// TIA Portal V20 export
TYPE "typeSequenceControlNode_GRnR"
// stored: Namespace Unit1.Em8
   STRUCT
      jobs : "LAF_typeJobs";
      sequence : "LAF_typeSequence";
      selectJobStatus { S7_SetPoint := 'True'} : Array[0..10] of "LAF_typeJobStatus";
      "step" : "LER_typeStep";
      jobInterface : "Unit1.Em8.typeSequenceControlNodeJobInterface_GRnR";
   END_STRUCT;
   // // "step".action1[101] : Step[101] : JOB[1] Condition
   // // "step".action1[110] : Step[110] : Hipot & Thickness Z-Axis Wait Pos
   // // "step".action1[111] : Step[111] : Servo Press Reference Home Pos
   // // "step".action1[120] : Step[120] : Tab Contactor Open
   // // "step".action1[121] : Step[121] : Tab Contactor Backward
   // // "step".action1[130] : Step[130] : Stage Lift Up
   // // "step".action1[140] : Step[140] : Spare
   // // "step".action1[150] : Step[150] : Stage Lift Down
   // // "step".action1[170] : Step[170] : Spare
   // // "step".action1[190] : Step[190] : JOB[1] Step End
   // // "step".action1[201] : Step[201] : JOB[2] Condition
   // // "step".action1[210] : Step[210] : Hipot & Thickness Loading Request => Transfer PP Left
   // // "step".action1[220] : Step[220] : Spare
   // // "step".action1[230] : Step[230] : Stage Lift Up
   // // "step".action1[240] : Step[240] : Hipot & Thickness Loading Check => Transfer PP Left
   // // "step".action1[250] : Step[250] : Spare
   // // "step".action1[290] : Step[290] : JOB[2] Step End
   // // "step".action1[301] : Step[301] : JOB[3] Condition
   // // "step".action1[310] : Step[310] : Stage Lift Down
   // // "step".action1[311] : Step[311] : Stage JR Detection Check
   // // "step".action1[320] : Step[320] : Spare
   // // "step".action1[330] : Step[330] : Press Start
   // // "step".action1[331] : Step[331] : Press Result
   // // "step".action1[340] : Step[340] : Thickness Z-Axis Thickness Ready Pos, Tab Forward
   // // "step".action1[341] : Step[341] : Thickness Z-Axis Measuring Thickness Pos, Tab Contactor Close
   // // "step".action1[350] : Step[350] : Thickness Start
   // // "step".action1[351] : Step[351] : Thickness Result
   // // "step".action1[352] : Step[352] : Thickness Z-Axis Wait Pos
   // // "step".action1[360] : Step[360] : Hipot Start
   // // "step".action1[361] : Step[361] : Hipot Result
   // // "step".action1[362] : Step[362] : Tab Contactor Open
   // // "step".action1[363] : Step[363] : Tab Contactor Backward
   // // "step".action1[380] : Step[380] : Press Home
   // // "step".action1[390] : Step[390] : JOB[3] Step End
   // // "step".action1[401] : Step[401] : JOB[4] Condition
   // // "step".action1[410] : Step[410] : Spare
   // // "step".action1[420] : Step[420] : Stage Lift Up
   // // "step".action1[430] : Step[430] : Hipot & Thickness Unloading Request => Transfer PP Right
   // // "step".action1[431] : Step[431] : Hipot & Thickness Unloading Check => Transfer PP Right
   // // "step".action1[480] : Step[480] : Stage Lift Down
   // // "step".action1[481] : Step[481] : Spare
   // // "step".action1[490] : Step[490] : JOB[4] Step End
   // // "step".transition1[101] : Step[101] : JOB[1] Condition
   // // "step".transition1[110] : Step[110] : Hipot & Thickness Z-Axis Wait Pos
   // // "step".transition1[111] : Step[111] : Servo Press Reference Home Pos
   // // "step".transition1[120] : Step[120] : Tab Contactor Open
   // // "step".transition1[121] : Step[121] : Tab Contactor Backward
   // // "step".transition1[130] : Step[130] : Stage Lift Up
   // // "step".transition1[140] : Step[140] : Spare
   // // "step".transition1[150] : Step[150] : Stage Lift Down
   // // "step".transition1[170] : Step[170] : Spare
   // // "step".transition1[190] : Step[190] : JOB[1] Step End
   // // "step".transition1[201] : Step[201] : JOB[2] Condition
   // // "step".transition1[210] : Step[210] : Hipot & Thickness Loading Request => Transfer PP Left
   // // "step".transition1[220] : Step[220] : Spare
   // // "step".transition1[230] : Step[230] : Stage Lift Up
   // // "step".transition1[240] : Step[240] : Hipot & Thickness Loading Check => Transfer PP Left
   // // "step".transition1[250] : Step[250] : Spare
   // // "step".transition1[290] : Step[290] : JOB[2] Step End
   // // "step".transition1[301] : Step[301] : JOB[3] Condition
   // // "step".transition1[310] : Step[310] : Stage Lift Down
   // // "step".transition1[311] : Step[311] : Stage JR Detection Check
   // // "step".transition1[320] : Step[320] : Spare
   // // "step".transition1[330] : Step[330] : Press Start
   // // "step".transition1[331] : Step[331] : Press Result
   // // "step".transition1[340] : Step[340] : Thickness Z-Axis Thickness Ready Pos, Tab Forward
   // // "step".transition1[341] : Step[341] : Thickness Z-Axis Measuring Thickness Pos, Tab Contactor Close
   // // "step".transition1[350] : Step[350] : Thickness Start
   // // "step".transition1[351] : Step[351] : Thickness Result
   // // "step".transition1[352] : Step[352] : Thickness Z-Axis Wait Pos
   // // "step".transition1[360] : Step[360] : Hipot Start
   // // "step".transition1[361] : Step[361] : Hipot Result
   // // "step".transition1[362] : Step[362] : Tab Contactor Open
   // // "step".transition1[363] : Step[363] : Tab Contactor Backward
   // // "step".transition1[380] : Step[380] : Press Home
   // // "step".transition1[390] : Step[390] : JOB[3] Step End
   // // "step".transition1[401] : Step[401] : JOB[4] Condition
   // // "step".transition1[410] : Step[410] : Spare
   // // "step".transition1[420] : Step[420] : Stage Lift Up
   // // "step".transition1[430] : Step[430] : Hipot & Thickness Unloading Request => Transfer PP Right
   // // "step".transition1[431] : Step[431] : Hipot & Thickness Unloading Check => Transfer PP Right
   // // "step".transition1[480] : Step[480] : Stage Lift Down
   // // "step".transition1[481] : Step[481] : Spare
   // // "step".transition1[490] : Step[490] : JOB[4] Step End
END_TYPE
